% RSLogix 500 project model_pressure_with_fans.RSS, saved by version 8.30.00.16 %
PROJECT "UNTITLED"    % processor: Bul.1763 MicroLogix 1100 Series B %

PROGRAM FILES
  LAD 2   3 rungs

DATA FILES
  O0 OUTPUT  4 elements
  I1 INPUT  6 elements
  S2 STATUS  66 elements
  B3 BINARY  1 elements
  T4 TIMER  1 elements
  C5 COUNTER  1 elements
  R6 CONTROL  1 elements
  N7 INTEGER  1 elements
  F8 FLOAT  15 elements

LADDER 2
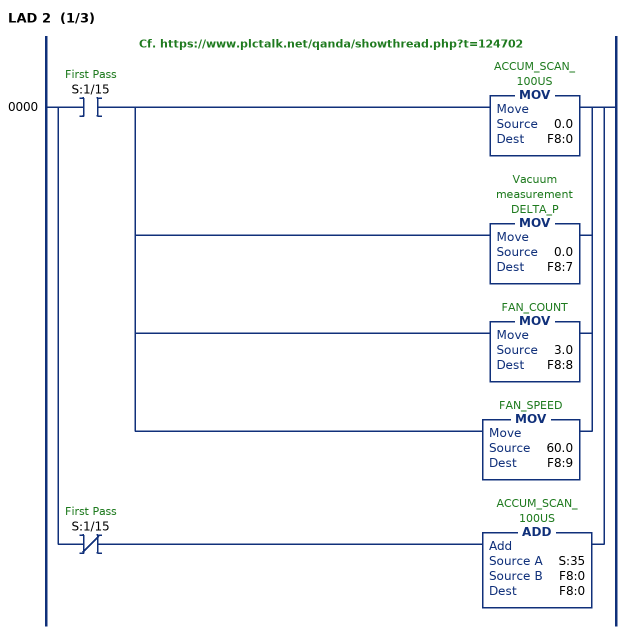
% Rung: 0 %
% TITLE: Cf. https://www.plctalk.net/qanda/showthread.php?t=124702 %
SOR BST XIC S:1/15 BST MOV 0.0 F8:0 NXB MOV 0.0 F8:7 NXB MOV 3.0 F8:8 NXB MOV 60.0 F8:9 BND NXB XIO S:1/15 ADD S:35 F8:0 F8:0 BND EOR
%   S:1/15  "First Pass" %
%   F8:0  ACCUM_SCAN_100US %
%   F8:7  DELTA_P  "Vacuum measurement" %
%   F8:8  FAN_COUNT %
%   F8:9  FAN_SPEED %
%   S:35  "Last 1 ms Scan Time" %

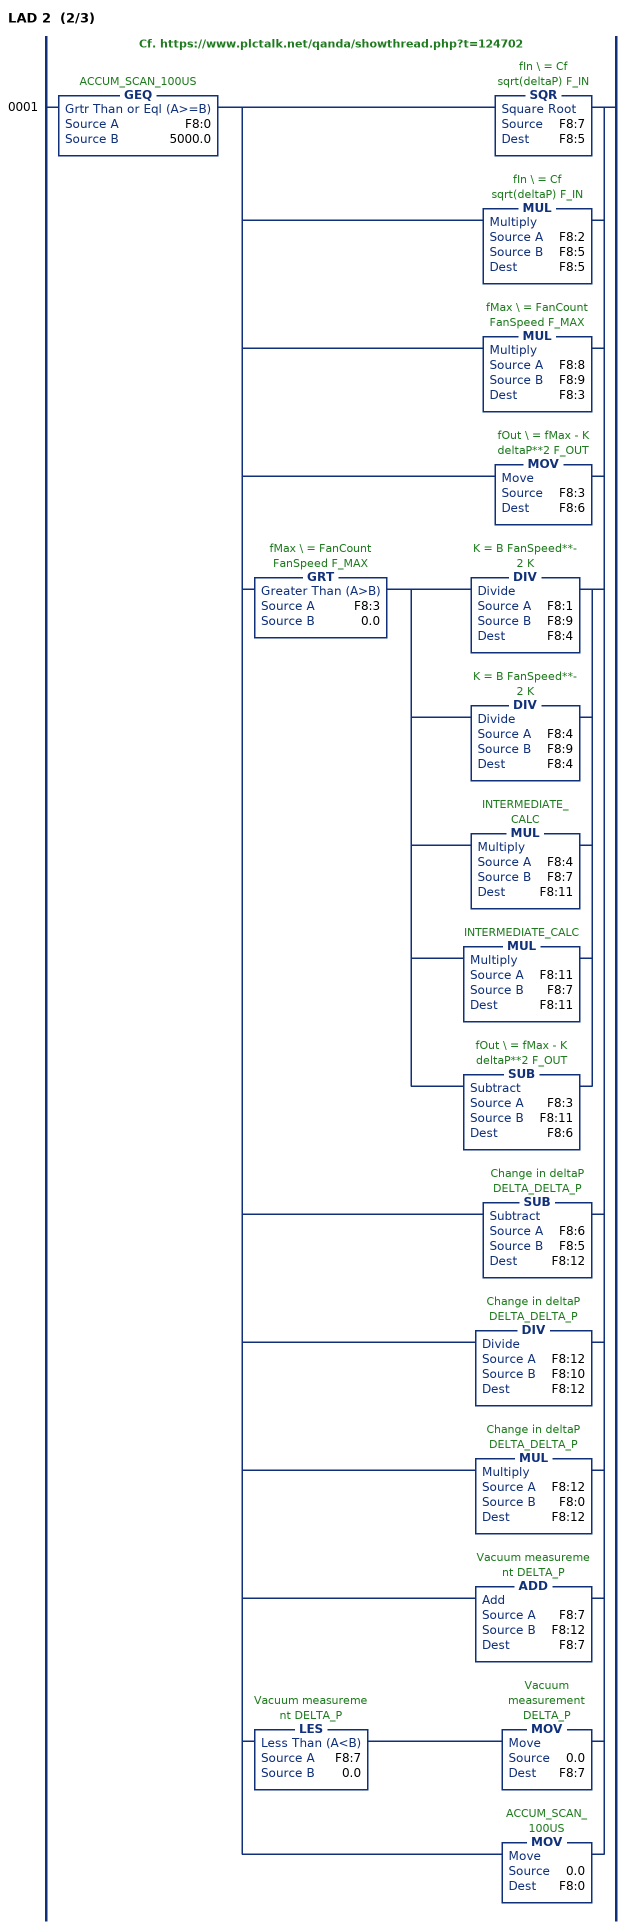
% Rung: 1 %
% TITLE: Cf. https://www.plctalk.net/qanda/showthread.php?t=124702 %
SOR GEQ F8:0 5000.0 BST SQR F8:7 F8:5 NXB MUL F8:2 F8:5 F8:5 NXB MUL F8:8 F8:9 F8:3 NXB MOV F8:3 F8:6 NXB GRT F8:3 0.0 BST DIV F8:1 F8:9 F8:4 NXB DIV F8:4 F8:9 F8:4 NXB MUL F8:4 F8:7 F8:11 NXB MUL F8:11 F8:7 F8:11 NXB SUB F8:3 F8:11 F8:6 BND NXB SUB F8:6 F8:5 F8:12 NXB DIV F8:12 F8:10 F8:12 NXB MUL F8:12 F8:0 F8:12 NXB ADD F8:7 F8:12 F8:7 NXB LES F8:7 0.0 MOV 0.0 F8:7 NXB MOV 0.0 F8:0 BND EOR
%   F8:0  ACCUM_SCAN_100US %
%   F8:7  DELTA_P  "Vacuum measurement" %
%   F8:5  F_IN  "fIn \ = Cf sqrt(deltaP)" %
%   F8:2  C_F  "Constant for K calc" %
%   F8:8  FAN_COUNT %
%   F8:9  FAN_SPEED %
%   F8:3  F_MAX  "fMax \ = FanCount FanSpeed" %
%   F8:6  F_OUT  "fOut \ = fMax - K deltaP**2" %
%   F8:1  B %
%   F8:4  K  "K = B FanSpeed**-2" %
%   F8:11  INTERMEDIATE_CALC %
%   F8:12  DELTA_DELTA_P  "Change in deltaP" %
%   F8:10  V  "Volume parameter" %

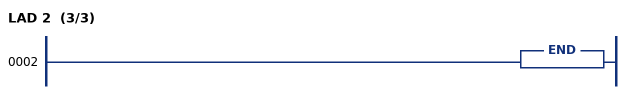
% Rung: 2 %
SOR END EOR

OTHER DOCUMENTED ADDRESSES
  FAN_COU  

DATA TABLE (non-zero values as saved)
DATA C5
% .PRE .ACC %
% C5:0 % 1000 0
DATA F8
% F8:0 % 0 18181.82 77.67989 0 0
% F8:10 % 1e+07 0 0 0 0
